INTERFACE I_ModbusSlave

PROPERTY Address : POINTER TO WORD
GET
END_GET
END_PROPERTY

METHOD Convert : BOOL
VAR_INPUT
	iRegionNo	:	INT;
	pReadData	:	POINTER TO BYTE;
END_VAR
END_METHOD

METHOD FirstCycle : BOOL
VAR_INPUT
END_VAR
END_METHOD

PROPERTY Name : STRING
GET
END_GET
SET
END_SET
END_PROPERTY

PROPERTY NumAddRegion : UINT
GET
END_GET
END_PROPERTY

PROPERTY UnitID : BYTE
GET
END_GET
SET
END_SET
END_PROPERTY

END_INTERFACE

(* stored: Version 1.1.0.1, ProductVersion 3.1.4024.12
   Itf I_ModbusSlave: Id {039c2ca5-0dea-4626-9cd9-3246cc113ed3}
   Property Address: Id {83375b69-0c0e-41fd-adcf-66c49f6a5589}
   Get Get: Id {d2b0a69c-7d10-479c-a1ef-8ff9feec14ac}
   Method Convert: Id {67b19cf7-dc69-4018-a62c-5d949742214d}
   Method FirstCycle: Id {cd0cef00-5605-4762-acf7-a002be0c2b78}
   Property Name: Id {9a85e90a-0671-41b2-b833-e0f20f4738bc}
   Get Get: Id {ca4c50f5-d11f-480a-8899-7122a5decbea}
   Set Set: Id {a14c142d-9121-4c38-b7ff-e77874b70c7e}
   Property NumAddRegion: Id {db368b18-d24b-45d2-a4ca-dcf7c2061b3a}
   Get Get: Id {4b55f151-f248-4743-8150-3137279a0323}
   Property UnitID: Id {0ee62372-dd01-418f-8379-ca4b49f91e15}
   Get Get: Id {a778e8f3-a6c5-4f14-8532-06abadf58f91}
   Set Set: Id {de016412-5d95-46cb-bfbe-b4d7cc6b9e03} *)
